FUNCTION_BLOCK FB_WriteOnChange
////////////////// 
// Write output variable , equals to input variable only if input variable changed state 
//////////////////	

VAR_INPUT
	Size			: UDINT; 				// Variable size 
	VarOut			: POINTER TO BYTE;		// Output  Variable Memory Address
	VarInput		: POINTER TO BYTE;		// Input Variable Memory Address	
END_VAR


VAR
	VarHold 		: DWORD  ; 	

END_VAR

IF MEMCMP(pBuf1:= VarInput, pBuf2:= ADR(VarHold) , n:=Size )<>0  THEN
	MEMCPY(srcAddr:= VarInput , destAddr := VarOut, n:= Size ) ;
END_IF

IF MEMCMP(pBuf1:= VarOut, pBuf2:= ADR(VarHold) , n:=Size )<>0  THEN
	MEMCPY(srcAddr:= VarOut , destAddr := VarInput, n:= Size ) ;
END_IF

MEMCPY(srcAddr:= VarInput , destAddr := ADR(VarHold), n:= Size ) ;

END_FUNCTION_BLOCK

(* stored: Version 1.1.0.1, ProductVersion 3.1.4024.6
   POU FB_WriteOnChange: Id {d85ba868-cd74-4a1c-aa28-456d76b70de2}, SpecialFunc None *)
